PROGRAM CraneCommander
VAR
	fTime : LREAL; 	
	bStarted : BOOL;
	fPosition : LREAL; 
	fInitialPosition : LREAL; 
	fInitialVelocity : LREAL; 
END_VAR

IF Inputs.bStart THEN
	fTime := fTime + Parameters.fCyclicTime;
ELSE
	fTime := 0; 	
END_IF

IF fTime > 0 THEN 
	bStarted := TRUE;
ELSE
	bStarted := FALSE;
END_IF

fPosition := Inputs.fVelocityReference * (fTime * fTime)/2 + fInitialVelocity * fTime + fInitialPosition;

Outputs.bSimulationStarted := bStarted;  
Outputs.fSimulationTime := fTime; 
Outputs.fCylinderVelocity := Inputs.fVelocityReference;

END_PROGRAM

(* stored: Version 1.1.0.1, ProductVersion 3.1.4024.9
   POU CraneCommander: Id {c255987f-7a58-4573-9ac9-545c12e8d4a5}, SpecialFunc None *)
